FUNCTION_BLOCK FB_MotionAxisHomeNC IMPLEMENTS I_MotionAxisHome
VAR
END_VAR

END_FUNCTION_BLOCK

(* stored: Version 1.1.0.1
   POU FB_MotionAxisHomeNC: Id {fe21bcc8-6662-4d7c-8885-dcc756df5d17}, SpecialFunc None *)
